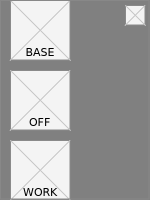
VISUALIZATION VisuCylinderVertDownCtrl  // 150x200
VAR_IN_OUT
	fbVisuCylinder: FB_VISU_CYLINDER;
END_VAR
    Rectangle (0,0 150x200)
    Image (10,140 60x60), "WORK", image: VisuSymbols.Symbols.TriangleDown
        OnMouseClick: execute {
            fbVisuCylinder.bMoveToBase:=FALSE;
            fbVisuCylinder.bMoveToWork:=true;
            fbVisuCylinder.bAllOff:=false;
            fbVisuCylinder.bFrameInvisible:= true;
        }
    Image (10,0 60x60), "BASE", image: VisuSymbols.Symbols.TriangleUp
        OnMouseClick: execute {
            fbVisuCylinder.bMoveToWork:=FALSE;
            fbVisuCylinder.bMoveToBase:=true;
            fbVisuCylinder.bAllOff:=false;
            fbVisuCylinder.bFrameInvisible:= true;
        }
    Image (125,5 20x20), image: VisuSymbols.Symbols.Wrong
        OnMouseDown: execute { fbVisuCylinder.bFrameInvisible:= true; }
    Image (10,70 60x60), "OFF", image: VisuSymbols.Symbols.Stop
        OnMouseClick: execute {
            fbVisuCylinder.bMoveToBase:=FALSE;
            fbVisuCylinder.bMoveToWork:=FALSE;
            fbVisuCylinder.bAllOff:=TRUE;
            fbVisuCylinder.bFrameInvisible:= true;
        }
END_VISUALIZATION

(* stored: Version 1.1.0.1, ProductVersion 3.1.4024.12
   Visu VisuCylinderVertDownCtrl: Id {2e8e55d6-cc8b-46ed-b8f4-2dd38a09ee13} *)
